// TIA Portal V17 export
// export: Created 2026-04-13T11:12:41.6982641Z, ExportSetting WithDefaults, DisplayName Totally Integrated Automation Portal, DisplayVersion V17 Update 4, DisplayName TIA Portal Openness, DisplayVersion V17 Update 4, DisplayName TIA Portal Version Control Interface, DisplayVersion V17, DisplayName SINAMICS Startdrive Advanced, DisplayVersion V17, DisplayName SINAMICS Startdrive G130, G150, S120, S150, SINAMICS MV, S210, DisplayVersion V17, DisplayName SINAMICS Startdrive G110M, G120, G120C, G120D, G120P, G115D, DisplayVersion V17, DisplayName STEP 7 Professional, DisplayVersion V17 Update 4, DisplayName STEP 7 Safety, DisplayVersion V17, DisplayName WinCC Professional, DisplayVersion V17 Update 4
FUNCTION_BLOCK "A8-报警功能块"   // FB13, SCL
{ S7_Optimized_Access := 'TRUE' }
VERSION : 0.1
// stored: AutoNumber true, IsIECCheckEnabled false, IsRetainMemResEnabled false, MemoryReserve 100, SetENOAutomatically false, UDAEnableTagReadback false
   VAR_INPUT
      报警0 : Bool;
      报警1 : Bool;
      报警2 : Bool;
      报警3 : Bool;
      报警4 : Bool;
      报警5 : Bool;
      报警6 : Bool;
      报警7 : Bool;
      报警8 : Bool;
      报警9 : Bool;
      报警10 : Bool;
      报警11 : Bool;
      报警12 : Bool;
      报警13 : Bool;
      报警14 : Bool;
      报警15 : Bool;
   END_VAR
   VAR
      报警 : Word;
      报警文本 : Array[0..15] of WString[20];
      off : Bool;
   END_VAR
BEGIN
    IF NOT  #off THEN

           #报警文本[0] := GetSymbolName(variable := #报警0, size := 0);
           #报警文本[1] := GetSymbolName(variable := #报警1, size := 0);
           #报警文本[2] := GetSymbolName(variable := #报警2, size := 0);
           #报警文本[3] := GetSymbolName(variable := #报警3, size := 0);
           #报警文本[4] := GetSymbolName(variable := #报警4, size := 0);
           #报警文本[5] := GetSymbolName(variable := #报警5, size := 0);
           #报警文本[6] := GetSymbolName(variable := #报警6, size := 0);
           #报警文本[7] := GetSymbolName(variable := #报警7, size := 0);

           #报警文本[8] := GetSymbolName(variable := #报警8, size := 0);
           #报警文本[9] := GetSymbolName(variable := #报警9, size := 0);
           #报警文本[10] := GetSymbolName(variable := #报警10, size := 0);
           #报警文本[11] := GetSymbolName(variable := #报警11, size := 0);
           #报警文本[12] := GetSymbolName(variable := #报警12, size := 0);
           #报警文本[13] := GetSymbolName(variable := #报警13, size := 0);
           #报警文本[14] := GetSymbolName(variable := #报警14, size := 0);
           #报警文本[15] := GetSymbolName(variable := #报警15, size := 0);

       END_IF;

       IF #报警0 THEN
           #报警.%X0 := 1;
       ELSE
           #报警.%X0 := 0;
       END_IF;

       IF #报警1 THEN
           #报警.%X1 := 1;
       ELSE
           #报警.%X1 := 0;
       END_IF;

       IF #报警2 THEN
           #报警.%X2 := 1;
       ELSE
           #报警.%X2 := 0;
       END_IF;


       IF #报警3 THEN
           #报警.%X3 := 1;
       ELSE
           #报警.%X3 := 0;
       END_IF;

       IF #报警4 THEN
           #报警.%X4 := 1;
       ELSE
           #报警.%X4 := 0;
       END_IF;

       IF #报警5 THEN
           #报警.%X5 := 1;
       ELSE
           #报警.%X5 := 0;
       END_IF;

       IF #报警6 THEN
           #报警.%X6 := 1;
       ELSE
           #报警.%X6 := 0;
       END_IF;

       IF #报警7 THEN
           #报警.%X7 := 1;
       ELSE
           #报警.%X7 := 0;
       END_IF;



       IF #报警8 THEN
           #报警.%X8 := 1;
       ELSE
           #报警.%X8 := 0;
       END_IF;

       IF #报警9 THEN
           #报警.%X9 := 1;
       ELSE
           #报警.%X9 := 0;
       END_IF;

       IF #报警10 THEN
           #报警.%X10 := 1;
       ELSE
           #报警.%X10 := 0;
       END_IF;


       IF #报警11 THEN
           #报警.%X11 := 1;
       ELSE
           #报警.%X11 := 0;
       END_IF;

       IF #报警12 THEN
           #报警.%X12 := 1;
       ELSE
           #报警.%X12 := 0;
       END_IF;

       IF #报警13 THEN
           #报警.%X13 := 1;
       ELSE
           #报警.%X13 := 0;
       END_IF;

       IF #报警14 THEN
           #报警.%X14 := 1;
       ELSE
           #报警.%X14 := 0;
       END_IF;

       IF #报警15 THEN
           #报警.%X15 := 1;
       ELSE
           #报警.%X15 := 0;
       END_IF;
END_FUNCTION_BLOCK
